(* PLC project CoDeSys External Library Template, WAGO e!COCKPIT e!COCKPIT, author 3S - Smart Software Solutions GmbH *)
(* stored: creationDateTime 2019-10-29T12:37:19.6302254, version 3.5.5.30, modificationDateTime 2019-10-29T12:36:39.3744516, organization 3S - Smart Software Solutions GmbH *)
(* Library project template with all possible element types, docu and a sample project structure *)

FUNCTION_BLOCK fbModbusDriverTCP
  VAR_INPUT
    intOdczytZapisZadanieRozmiarBufora : INT;
    arTCPParametryKomunikacji : typModbusTCPParametryKomunikacji;
  END_VAR
  VAR_IN_OUT
    arOdczytCykliczny : ARRAY[1..1000] OF typModbusOdczytCykliczny;
    arOdczytZapisZadanie : ARRAY[1..1000] OF typModbusOdczytZapisZadanie;
    arStatusKomunikacji : ARRAY[1..256] OF INT;
    intZnacznikOdczytuZapisuZadanie : INT;
  END_VAR
  VAR
    ModbusMasterTCP : FbMbMasterTcp;
    utZapytanie : typMBQuery;
    utOdpowiedz : typMbResponse;
    xStatusPolaczenia : BOOL;
    xBladKomunikacji : BOOL;
    typStatusKomunikacji : WagoSysErrorBase.FbResult;
    fbTimerRestartuPolaczenia : TON;
    tCzasRestartuPolaczenia : TIME := TIME#15s0ms;
    tCzasPonowienia : LTIME := LTIME#15s0ms0us0ns;
    tCzasStabilnosciKomunikacji : LTIME := LTIME#30s0ms0us0ns;  (* czas po jakim driver raportuje poprawną komunikację po jej faktycznym odzyskaniu - czas powinien być większy niż czas tCzasPonawiania *)
    xDriverWykonajKomunikacje : BOOL;
    arStatusKomunikacjiTimestampOstatniaProba : ARRAY[1..256] OF LTIME;
    arStatusKomunikacjiTimestampOstatniBlad : ARRAY[1..256] OF LTIME;
    negWykonaj : F_TRIG;
    intZnacznikDriveraOdczytuCyklicznego : INT := 1;
    intZnacznikDriveraOdczytuZapisuZadanie : INT := 1;
    intZnacznikOdczytuCyklicznegoReferencja : INT;
    intZnacznikOdczytuCyklicznegoPoczatek : INT;
    intZnacznikOdczytuZapisuZadanieReferencja : INT;
    intZnacznikPomocniczy : INT;
    intOdczytZadanieTablica : INT;
    intOdczytCyklicznyTablica : INT;
    intOdczytCyklicznyTablicaIlosc : INT;
    intLoop : INT;
    intDebugZnacznik : INT;  (* debug *)
    arDebugZapytanie : ARRAY[0..1000] OF typMBQuery;
    arDebugOdpowiedz : ARRAY[0..1000] OF typMbResponse;
    typDebugOdczytZapisZadanie : ARRAY[0..1000] OF typModbusOdczytZapisZadanie;
    arDebugCzas : ARRAY[0..1000] OF DT;
  END_VAR

            // obsługa odczytu zapisu danych na żądanie

IF intZnacznikDriveraOdczytuZapisuZadanie <> intZnacznikOdczytuZapisuZadanie AND NOT xDriverWykonajKomunikacje THEN
	fnTablicaKomunikatowInkrementacja(intRozmiarTablicy := intOdczytZapisZadanieRozmiarBufora, intWskaznik := intZnacznikDriveraOdczytuZapisuZadanie);
	IF arStatusKomunikacji[arOdczytZapisZadanie[intZnacznikDriveraOdczytuZapisuZadanie].bAdresUrzadzenia] = enumModbusStatus.KomunikacjaPrawidlowa  AND xStatusPolaczenia THEN
		xDriverWykonajKomunikacje := TRUE;
		utZapytanie.bUnitId := arOdczytZapisZadanie[intZnacznikDriveraOdczytuZapisuZadanie].bAdresUrzadzenia;
		utZapytanie.bFunctionCode := arOdczytZapisZadanie[intZnacznikDriveraOdczytuZapisuZadanie].bFunkcja;
		utZapytanie.uiReadQuantity := 1;
		utZapytanie.uiReadAddress := arOdczytZapisZadanie[intZnacznikDriveraOdczytuZapisuZadanie].uiAdresRejestru;
		utZapytanie.uiWriteAddress := arOdczytZapisZadanie[intZnacznikDriveraOdczytuZapisuZadanie].uiAdresRejestru;
		utZapytanie.awWriteData[0] := arOdczytZapisZadanie[intZnacznikDriveraOdczytuZapisuZadanie].wWartoscDoZapisania;
		utZapytanie.uiWriteQuantity := 1;
		intOdczytZadanieTablica := intZnacznikDriveraOdczytuZapisuZadanie;
	END_IF
END_IF

// obsługa odczytu zmiennych zapisanych w tabeli

IF NOT xDriverWykonajKomunikacje AND xStatusPolaczenia AND NOT xBladKomunikacji THEN

	intZnacznikOdczytuCyklicznegoReferencja := intZnacznikDriveraOdczytuCyklicznego;
	intZnacznikDriveraOdczytuCyklicznego := intZnacznikDriveraOdczytuCyklicznego + 1;
	IF arOdczytCykliczny[intZnacznikDriveraOdczytuCyklicznego].bAdresUrzadzenia = 0 THEN
		intZnacznikDriveraOdczytuCyklicznego := 1;
	END_IF

	WHILE intZnacznikOdczytuCyklicznegoReferencja <> intZnacznikDriveraOdczytuCyklicznego AND _GetLongTime() - arStatusKomunikacjiTimestampOstatniaProba[arOdczytCykliczny[intZnacznikDriveraOdczytuCyklicznego].bAdresUrzadzenia] < tCzasPonowienia AND
			_GetLongTime() - arOdczytCykliczny[intZnacznikDriveraOdczytuCyklicznego].ltZnacznikCzasuWyslania < arOdczytCykliczny[intZnacznikDriveraOdczytuCyklicznego].ltCzestotliwosc DO
		intZnacznikDriveraOdczytuCyklicznego := intZnacznikDriveraOdczytuCyklicznego + 1;
		IF arOdczytCykliczny[intZnacznikDriveraOdczytuCyklicznego].bAdresUrzadzenia = 0 THEN
			intZnacznikDriveraOdczytuCyklicznego := 1;
		END_IF
	END_WHILE

// zapis adresu startowego rejestrów do zapisu

	IF intZnacznikOdczytuCyklicznegoReferencja <> intZnacznikDriveraOdczytuCyklicznego THEN
		xDriverWykonajKomunikacje := TRUE;
		arStatusKomunikacjiTimestampOstatniaProba[arOdczytCykliczny[intZnacznikDriveraOdczytuCyklicznego].bAdresUrzadzenia] := _GetLongTime();
		utZapytanie.bUnitId := arOdczytCykliczny[intZnacznikDriveraOdczytuCyklicznego].bAdresUrzadzenia;
		utZapytanie.bFunctionCode := arOdczytCykliczny[intZnacznikDriveraOdczytuCyklicznego].bFunkcja;
		utZapytanie.uiReadAddress := arOdczytCykliczny[intZnacznikDriveraOdczytuCyklicznego].uiAdresRejestru;
		utZapytanie.uiReadQuantity := 1;
		intOdczytCyklicznyTablica := intZnacznikDriveraOdczytuCyklicznego;
		intZnacznikOdczytuCyklicznegoReferencja := intZnacznikDriveraOdczytuCyklicznego;
		intZnacznikPomocniczy := intZnacznikDriveraOdczytuCyklicznego + 1;
		IF arOdczytCykliczny[intZnacznikPomocniczy].bAdresUrzadzenia = 0 THEN
			intZnacznikPomocniczy := 1;
		END_IF

// sprawdzenie czy następne żądanie nie jest w kolejności do bieżącego jeśli tak to grupuje je w jedno zapytanie

		WHILE (arOdczytCykliczny[intZnacznikPomocniczy].uiAdresRejestru - arOdczytCykliczny[intZnacznikDriveraOdczytuCyklicznego].uiAdresRejestru = 1 AND
				arOdczytCykliczny[intZnacznikPomocniczy].bFunkcja = arOdczytCykliczny[intZnacznikDriveraOdczytuCyklicznego].bFunkcja AND
				arOdczytCykliczny[intZnacznikPomocniczy].bAdresUrzadzenia = arOdczytCykliczny[intZnacznikDriveraOdczytuCyklicznego].bAdresUrzadzenia) DO
				
			utZapytanie.uiReadQuantity := utZapytanie.uiReadQuantity + 1;
			intZnacznikDriveraOdczytuCyklicznego := intZnacznikDriveraOdczytuCyklicznego + 1;
			IF arOdczytCykliczny[intZnacznikDriveraOdczytuCyklicznego].bAdresUrzadzenia = 0 THEN
				intZnacznikDriveraOdczytuCyklicznego := 1;
			END_IF
			intZnacznikPomocniczy := intZnacznikDriveraOdczytuCyklicznego + 1;
			IF arOdczytCykliczny[intZnacznikPomocniczy].bAdresUrzadzenia = 0 THEN
				intZnacznikPomocniczy := 1;
			END_IF
		END_WHILE
		intOdczytCyklicznyTablicaIlosc := UINT_TO_INT(utZapytanie.uiReadQuantity);
	END_IF
END_IF

// restart połączenia jeśli brak komunikacji

fbTimerRestartuPolaczenia(IN := (NOT xStatusPolaczenia OR xBladKomunikacji) AND NOT fbTimerRestartuPolaczenia.Q, PT := tCzasRestartuPolaczenia);

// driver komunikacyjny MODBUS TCP

ModbusMasterTCP(xConnect :=			NOT fbTimerRestartuPolaczenia.Q ,
				sHost :=			arTCPParametryKomunikacji.sAdresTCP ,
				wPort := 			arTCPParametryKomunikacji.wPortTCP ,
				utKeepAlive := 		arTCPParametryKomunikacji.utPodtrzymajWtyczkeTCP ,
				eFrameType := 		arTCPParametryKomunikacji.eTypRamki ,
				tTimeOut := 		arTCPParametryKomunikacji.tTimeOut ,
					
				xIsOpen => 			xStatusPolaczenia ,
				xError => 			xBladKomunikacji ,
				oStatus => 			typStatusKomunikacji ,
					
				xTrigger := 		xDriverWykonajKomunikacje , 
				utQuery := 			utZapytanie , 
				utResponse := 		utOdpowiedz);

// obługa akcji po zakończeniu zadania komunikacji (zapis wartości , zapis błędu itd)
	
negWykonaj(CLK := xDriverWykonajKomunikacje);

IF negWykonaj.Q THEN
// jeżeli był błąd komunikacji wpisz go do tablicy błędów

	IF xBladKomunikacji THEN
		arStatusKomunikacji[utZapytanie.bUnitId] := enumModbusStatus.BrakKomunikacji;
		arStatusKomunikacjiTimestampOstatniBlad[utZapytanie.bUnitId] := _GetLongTime();
		ELSE
		IF _GetLongTime() - arStatusKomunikacjiTimestampOstatniBlad[utZapytanie.bUnitId] > tCzasStabilnosciKomunikacji AND arStatusKomunikacji[utZapytanie.bUnitId] <> enumModbusStatus.KomunikacjaPrawidlowa THEN	
			arStatusKomunikacji[utZapytanie.bUnitId] := enumModbusStatus.KomunikacjaPrawidlowa;
		END_IF

// jeżeli zapytanie było żądaniem  wysłania danych

		IF utZapytanie.bFunctionCode = enumModbusKodyFunkcji.OdczytWejscBitowych OR utZapytanie.bFunctionCode = enumModbusKodyFunkcji.OdczytWyjscBitowych OR
			utZapytanie.bFunctionCode = enumModbusKodyFunkcji.OdczytNRejestrow OR utZapytanie.bFunctionCode = enumModbusKodyFunkcji.OdczytNRejestrowWejsciowych THEN
			intZnacznikOdczytuCyklicznegoPoczatek := 0;
		
// jeżeli był wykonany rozkaz odczytu danych z cyklu "na żądanie"

			IF intOdczytZadanieTablica <> 0 THEN
				arDebugZapytanie[intDebugZnacznik] := utZapytanie;
				arDebugOdpowiedz[intDebugZnacznik] := utOdpowiedz;
				typDebugOdczytZapisZadanie[intDebugZnacznik] := arOdczytZapisZadanie[intZnacznikDriveraOdczytuZapisuZadanie];				
				arDebugCzas[intDebugZnacznik] := FuGetDateAndTime();
				fnTablicaKomunikatowInkrementacja(intRozmiarTablicy := 900, intWskaznik := intDebugZnacznik);
//				arOdczytZapisZadanie[intZnacznikDriveraOdczytuZapisuZadanie].pZmiennaDoOdczytu^ := utOdpowiedz.awData[0];
			END_IF

// jeżeli był wykonany rozkaz odczytu danych z cyklu "cykliczny"

			IF intOdczytCyklicznyTablica <> 0 THEN
				FOR intLoop := 1 TO intOdczytCyklicznyTablicaIlosc DO
					arOdczytCykliczny[intOdczytCyklicznyTablica + intLoop - 1].pZmiennaReferencyjna^ := utOdpowiedz.awData[intLoop - 1];
					arOdczytCykliczny[intOdczytCyklicznyTablica + intLoop - 1].ltZnacznikCzasuWyslania := _GetLongTime();
				END_FOR
			END_IF
		END_IF
	END_IF
	intOdczytZadanieTablica := 0;
	intOdczytCyklicznyTablica := 0;
	intOdczytCyklicznyTablicaIlosc := 0;
END_IF
          
END_FUNCTION_BLOCK
